TYPE ST_CART :
STRUCT
	nNAME: STRING;
	posX:INT;
	posY:INT;
	color:INT;
	position: INT;
END_STRUCT
END_TYPE

(* stored: Version 1.1.0.1, ProductVersion 3.1.4024.12
   DUT ST_CART: Id {3456120e-8460-4c6c-bd03-2d96c3a966e0} *)
